DATA_BLOCK "DB7_TRAZA"
{ S7_Optimized_Access := 'TRUE' }
VERSION : 0.1
NON_RETAIN
   VAR RETAIN
      Gestion { S7_SetPoint := 'False'} : "UDT_ZC_TRAZA_GESTION";
      Registro { S7_SetPoint := 'False'} : "UDT_ZC_TRAZA_DATOS";
      Buffer { S7_SetPoint := 'False'} : Array[0.."N_MAX_TRAZA_BUFFER"] of "UDT_ZC_TRAZA_DATOS";
   END_VAR


BEGIN
   Gestion.HabilitacionGeneral := TRUE;
   Gestion.EstadoConexion := TRUE;
   Gestion.OrdenIniciar := FALSE;
   Gestion.HabilitarCategoria[1] := TRUE;
   Gestion.HabilitarCategoria[2] := FALSE;
   Gestion.HabilitarCategoria[3] := TRUE;
   Gestion.HabilitarCategoria[4] := FALSE;
   Gestion.HabilitarCategoria[5] := FALSE;
   Gestion.HabilitarCategoria[6] := FALSE;
   Gestion.HabilitarCategoria[7] := FALSE;
   Gestion.HabilitarCategoria[8] := FALSE;
   Gestion.HabilitarCategoria[9] := FALSE;
   Gestion.HabilitarCategoria[10] := FALSE;
   Gestion.HabilitarCategoria[11] := FALSE;
   Gestion.HabilitarCategoria[12] := FALSE;
   Gestion.HabilitarCategoria[13] := FALSE;
   Gestion.HabilitarCategoria[14] := FALSE;
   Gestion.HabilitarCategoria[15] := FALSE;
   Gestion.Etapa := 0;
   Gestion.SP_Tiempo := 2;
   Gestion.TiempoActual := 0;
   Registro.Registrar := 0;
   Registro.TimeStamp := '';
   Registro.Categoria := 0;
   Registro.User := '';
   Registro.Texto := '';
   Buffer[0].Registrar := 0;
   Buffer[0].TimeStamp := '';
   Buffer[0].Categoria := 0;
   Buffer[0].User := '';
   Buffer[0].Texto := '';
   Buffer[1].Registrar := 0;
   Buffer[1].TimeStamp := '';
   Buffer[1].Categoria := 0;
   Buffer[1].User := '';
   Buffer[1].Texto := '';
   Buffer[2].Registrar := 0;
   Buffer[2].TimeStamp := '';
   Buffer[2].Categoria := 0;
   Buffer[2].User := '';
   Buffer[2].Texto := '';
   Buffer[3].Registrar := 0;
   Buffer[3].TimeStamp := '';
   Buffer[3].Categoria := 0;
   Buffer[3].User := '';
   Buffer[3].Texto := '';
   Buffer[4].Registrar := 0;
   Buffer[4].TimeStamp := '';
   Buffer[4].Categoria := 0;
   Buffer[4].User := '';
   Buffer[4].Texto := '';
   Buffer[5].Registrar := 0;
   Buffer[5].TimeStamp := '';
   Buffer[5].Categoria := 0;
   Buffer[5].User := '';
   Buffer[5].Texto := '';
   Buffer[6].Registrar := 0;
   Buffer[6].TimeStamp := '';
   Buffer[6].Categoria := 0;
   Buffer[6].User := '';
   Buffer[6].Texto := '';
   Buffer[7].Registrar := 0;
   Buffer[7].TimeStamp := '';
   Buffer[7].Categoria := 0;
   Buffer[7].User := '';
   Buffer[7].Texto := '';
   Buffer[8].Registrar := 0;
   Buffer[8].TimeStamp := '';
   Buffer[8].Categoria := 0;
   Buffer[8].User := '';
   Buffer[8].Texto := '';
   Buffer[9].Registrar := 0;
   Buffer[9].TimeStamp := '';
   Buffer[9].Categoria := 0;
   Buffer[9].User := '';
   Buffer[9].Texto := '';
   Buffer[10].Registrar := 0;
   Buffer[10].TimeStamp := '';
   Buffer[10].Categoria := 0;
   Buffer[10].User := '';
   Buffer[10].Texto := '';
   Buffer[11].Registrar := 0;
   Buffer[11].TimeStamp := '';
   Buffer[11].Categoria := 0;
   Buffer[11].User := '';
   Buffer[11].Texto := '';
   Buffer[12].Registrar := 0;
   Buffer[12].TimeStamp := '';
   Buffer[12].Categoria := 0;
   Buffer[12].User := '';
   Buffer[12].Texto := '';
   Buffer[13].Registrar := 0;
   Buffer[13].TimeStamp := '';
   Buffer[13].Categoria := 0;
   Buffer[13].User := '';
   Buffer[13].Texto := '';
   Buffer[14].Registrar := 0;
   Buffer[14].TimeStamp := '';
   Buffer[14].Categoria := 0;
   Buffer[14].User := '';
   Buffer[14].Texto := '';
   Buffer[15].Registrar := 0;
   Buffer[15].TimeStamp := '';
   Buffer[15].Categoria := 0;
   Buffer[15].User := '';
   Buffer[15].Texto := '';

END_DATA_BLOCK

